# B&R Automation Studio project Ionova-Pobedrya-SW-MaRS-Lab1
Automation Studio 

## Logical view

### Library Logical/Libraries/MotorCtrl

#### MotorCtrl.fun
```iecst
{REDUND_OK} FUNCTION_BLOCK FB_Integrator (*Integrator function block*) (*$GROUP=User,$CAT=User,$GROUPICON=User.png,$CATICON=User.png*)
	VAR_INPUT
		in : REAL; (*integrator input*)
	END_VAR
	VAR_OUTPUT
		out : REAL; (*integrator output*)
	END_VAR
	VAR
		dt : REAL; (*step [s]*)
	END_VAR
END_FUNCTION_BLOCK

{REDUND_OK} FUNCTION_BLOCK FB_Motor (*Motor function block*) (*$GROUP=User,$CAT=User,$GROUPICON=User.png,$CATICON=User.png*)
	VAR_INPUT
		u : REAL; (*input voltage [V]*)
	END_VAR
	VAR_OUTPUT
		phi : REAL; (*rotation frequency [rpm]*)
		w : REAL; (*position [rad]*)
	END_VAR
	VAR
		integrator : FB_Integrator; (*integrator*)
		Tm : REAL; (*electromechanical time constant*)
		ke : REAL; (*motor EMF constant [V/rpm] *)
		dt : REAL; (*step [s]*)
	END_VAR
END_FUNCTION_BLOCK

{REDUND_OK} FUNCTION_BLOCK FB_Regulator (*Regulator function block*) (*$GROUP=User,$CAT=User,$GROUPICON=User.png,$CATICON=User.png*)
	VAR_INPUT
		e : REAL; (*Error between input and real frequency [rpm]*)
	END_VAR
	VAR_OUTPUT
		u : REAL; (*input voltage [V]*)
	END_VAR
	VAR
		k_p : REAL; (*proportional gain*)
		k_i : REAL; (*integral gain*)
		integrator : FB_Integrator; (*integrator*)
		iyOld : REAL; (*stores the prev value of the anti-accumulation system*)
		max_abs_value : REAL; (*limit block max value [V]*)
		dt : REAL; (*step [s]*)
		e_p : USINT; (*temporary variable*)
	END_VAR
END_FUNCTION_BLOCK
```

#### FB_Integrator.c
```c
#include <bur/plctypes.h>
#ifdef __cplusplus
	extern "C"
	{
#endif
	#include "MotorCtrl.h"
#ifdef __cplusplus
	};
#endif
/* integrator */
void FB_Integrator(struct FB_Integrator* inst)
{
	inst->out += inst->in;
}
```

#### FB_Motor.c
```c
#include <bur/plctypes.h>
#ifdef __cplusplus
	extern "C"
	{
#endif
	#include "MotorCtrl.h"
#ifdef __cplusplus
	};
#endif
/* motor */
void FB_Motor(struct FB_Motor* inst)
{

	{
	inst->integrator.in = (inst->u*(1/inst->ke) -inst->w)*(inst->dt/inst->Tm);
	FB_Integrator(&(inst->integrator));
	inst->w = inst->integrator.out;
	inst->integrator.in = inst->w*inst->dt;
	FB_Integrator(&(inst->integrator));
	inst->phi = inst->integrator.out;
	}
}
```

#### FB_Regulator.c
```c
#include <bur/plctypes.h>
#ifdef __cplusplus
	extern "C"
	{
#endif
	#include "MotorCtrl.h"
#ifdef __cplusplus
	};
#endif

void FB_Regulator(struct FB_Regulator* inst)
{

	inst->integrator.in = inst->iyOld + inst->e * inst->k_i * inst->dt;
	FB_Integrator(&(inst->integrator));

	inst->e_p = inst->e*inst->k_p;

	if(inst->e_p < inst->max_abs_value || inst->e_p > -inst->e_p > -inst->max_abs_value);
	else
	{
		if(inst->e_p>0) inst->e_p = inst->max_abs_value;
		else inst->e_p = -inst->max_abs_value;
	}

	inst->e_p += inst->integrator.out;

	if(inst->e_p < inst->max_abs_value || inst->e_p > -inst->e_p > -inst->max_abs_value)
		inst->u = inst->e_p;
	else
	{
		if(inst->e_p>0) inst->u = inst->max_abs_value;
		else inst->u = -inst->max_abs_value;
	}

	inst->iyOld = inst->u - inst->e_p;

}
```

### Program Logical/Program

#### Variables.var
```iecst
VAR
	Speed : REAL;
	Enable : BOOL;
	fb_motor_1 : FB_Motor;
	fb_motor_2 : FB_Motor;
	fb_regulator : FB_Regulator;
	counter : REAL;
END_VAR
```

#### Cyclic.c
```c
#include <bur/plctypes.h>

#ifdef _DEFAULT_INCLUDES
	#include <AsDefault.h>
#endif

void _CYCLIC ProgramCyclic(void)
{

	if (Enable == 1)
	{
		counter += 1;
		if (counter >= 10000 && counter <= 15000) Speed = 5;
		else Speed = 0;
	}
	else Speed = 0;

	fb_regulator.e = Speed - fb_motor_1.w;
	FB_Regulator(&(fb_regulator));
	fb_motor_1.u = fb_regulator.u*fb_motor_1.ke;
	fb_motor_2.u = Speed*fb_motor_2.ke;
	FB_Motor(&(fb_motor_1));
	FB_Motor(&(fb_motor_2));

}
```

#### Init.c
```c
#include <bur/plctypes.h>

#ifdef _DEFAULT_INCLUDES
	#include <AsDefault.h>
#endif

void _INIT ProgramInit(void)
{
	Enable = 1;
	counter = 0;
	Speed = 0;

	fb_regulator.dt = 0.02;
	fb_regulator.k_i = 16;
	fb_regulator.k_p = 0.64;
	fb_regulator.max_abs_value = 24;

	fb_motor_1.dt = 0.02;
	fb_motor_1.ke = 16;
	fb_motor_1.Tm = 0.04;

	fb_motor_2.dt = 0.02;
	fb_motor_2.ke = 16;
	fb_motor_2.Tm = 0.04;
}
```
